FUNCTION_BLOCK FB_CRYO_LN2_CTRL EXTENDS FB_CRYO_BIN_CTRL
VAR_INPUT
	in_lrTempK:		LREAL;			// Temperature input value [K]
	in_bValid:		BOOL := TRUE;	// Temperature Valid flag
	// Two parameters for decision making
	in_lrTempValveOpen:		LREAL := 91.27;		// Open  valve if temperature above this value [K]
	in_lrTempValveClose:	LREAL := 79.148;	// Close valve if temperature below this value [K]
END_VAR
VAR_OUTPUT
END_VAR
VAR
END_VAR

// Check the validity of the temperature reading.
// Start the check after 200 cycles.
IF stat.nCycleCounter > 200 THEN
	IF NOT in_bValid THEN
		// The temperature is not valid. 
		// The controller cannot work.
		stat.bCtrlOK	:= FALSE;
	ELSIF in_lrTempValveClose >= in_lrTempValveOpen THEN
		// Wrong configuration.
		// ValveClose MUST be lower than ValveOpen temperature
		stat.bCtrlOK	:= FALSE;
	ELSE
		// The temperature is valid. 
		stat.bCtrlOK	:= TRUE;
	END_IF
ELSE
	// The temperature is valid. 
	stat.bCtrlOK	:= TRUE;
END_IF

// Execute parent FB.
SUPER^();

METHOD M_SetStatus
VAR_INPUT
	nState:	E_CRYO_BIN_CTRL_STATE;
END_VAR
// Execute the status of the parent FB
SUPER^.M_SetStatus(nState);

// Set proper error description, if any.
IF Actuator.stat.bError THEN
	stat.sState	:= 'Valve failure';
ELSIF NOT stat.bCtrlOK THEN
	stat.sState	:= 'Temperature not valid';
END_IF
END_METHOD

METHOD M_User_SetAction : INT
VAR_INPUT
END_VAR
// TODO USER
// Overwrite Method FB_CRYO_BIN_CTRL::M_User_SetOutput()
//
// This method implements the logic for controlling the LN2 valve.
// 
// FB_CRYO_LN2_CTRL input parameters:
//
// in_lrTempK          - LN2 temperature
// in_bValid           - Flag if temperature reading is valid
// in_lrTempValveOpen  - Temperature upper limit [K]. Valve opens  when:  LN2 > in_lrTempValveOpen
// in_lrTempValveClose - Temperature lower limit [K]. Valve closes when:  LN2 < in_lrTempValveClose
//
// in_lrTempValveOpen > in_lrTempValveClose, e.g. 91.27K > 79.148K.
//
	
IF	stat.nState = E_CRYO_BIN_CTRL_STATE.ACTIVE_OFF  OR  
	stat.nState = E_CRYO_BIN_CTRL_STATE.ACTIVE_ON THEN
	// Check if input temperature value is valid.
	// If OK, check temperature against the limits	
	IF NOT stat.bCtrlOK THEN
		// Temperature reading is not valid.
		// Dectivate the actuator, i.e. close the valve
		M_User_SetAction	:= E_CRYO_BIN_CTRL_ACTION.OFF;
		stat.nState	:= E_CRYO_BIN_CTRL_STATE.ERROR;
	ELSIF in_lrTempK > in_lrTempValveOpen THEN
		// Activate the actuator, i.e. open the valve
		M_User_SetAction	:= E_CRYO_BIN_CTRL_ACTION.ON;
	ELSIF in_lrTempK < in_lrTempValveClose THEN
		// Dectivate the actuator, i.e. close the valve
		M_User_SetAction	:= E_CRYO_BIN_CTRL_ACTION.OFF;
	END_IF
	
ELSE
	// Don't do anything
	M_User_SetAction	:= E_CRYO_BIN_CTRL_ACTION.NONE;
END_IF
END_METHOD

END_FUNCTION_BLOCK

(* stored: Version 1.1.0.1, ProductVersion 3.1.4024.9
   POU FB_CRYO_LN2_CTRL: Id {66ff87ce-ff5b-4d3a-9b1b-9ce460018a96}, SpecialFunc None
   Method M_SetStatus: Id {5a1cfb82-a4d3-4622-9494-80a373e92cbf}
   Method M_User_SetAction: Id {d02b2084-6399-4480-99c9-a37797d8dc6c} *)
